{attribute 'qualified_only'}
{attribute 'strict'}
TYPE AxisFunctions :
(
	enum_member := 0
);
END_TYPE

(* stored: Version 1.1.0.1, ProductVersion 3.1.4022.10
   EnumerationTextList AxisFunctions: Id {5cd32b0e-ae25-4cef-a6fd-83fa9e4daaf4} *)
